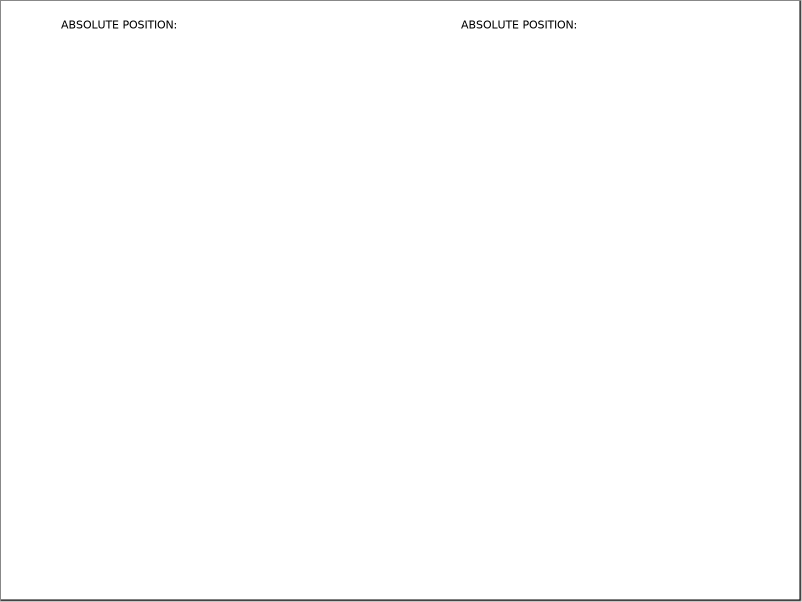
VISUALIZATION F05_Read_Parameter  // 802x602
    Rectangle (0,0 800x600)
    Label (10,10 170x30), "ABSOLUTE POSITION:"
    Label (410,10 170x30), "ABSOLUTE POSITION:"
END_VISUALIZATION

(* stored: Version 1.1.0.1, ProductVersion 3.1.4022.7
   Visu F05_Read_Parameter: Id {64b8fcc4-d5fc-4fa0-ba5e-2d2f48312d1f} *)
